INTERFACE I_Logger

METHOD PUBLIC M_Attach : BOOL
VAR_INPUT
	iLogging:				I_Logger;
END_VAR
END_METHOD

METHOD PUBLIC M_Log : BOOL
VAR_INPUT
	stMessage:			ST_Message;
END_VAR
END_METHOD

PROPERTY PUBLIC P_LogLevel : E_LogLevel
GET
END_GET
SET
END_SET
END_PROPERTY

END_INTERFACE

(* stored: Version 1.1.0.1
   Itf I_Logger: Id {c8546c00-1964-4def-86cd-48ddf720fa88}
   Method M_Attach: Id {d8504e1d-ba05-46db-8e36-f183866560d7}
   Method M_Log: Id {70349284-7301-41be-b202-535da7461a8a}
   Property P_LogLevel: Id {f99cbbda-76c9-45bd-bfff-f0a515bcf17d}
   Get Get: Id {7944be96-fe0f-454d-b80e-0d57feb93034}
   Set Set: Id {629baaa2-9d8b-4230-8de8-dc02daae734e} *)
